// TIA Portal V18 export
FUNCTION "fcFonctionMathLAD" : Void   // FC7, LAD
{ S7_Optimized_Access := 'TRUE' }
// stored: SetENOAutomatically false
   VAR_INPUT
      iInput1 : Bool;
      iInput2 : Bool;
      iInput3 : Bool;
   END_VAR
   VAR_OUTPUT
      oOutput : Bool;
   END_VAR
BEGIN

REGION Network 1
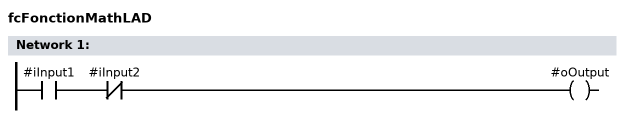
   RUNG wire#powerrail
      Contact( #iInput1 )
      I_Contact( #iInput2 )
      Coil( #oOutput )
   END_RUNG
   // the same network as SCL:
   #oOutput := #iInput1 AND NOT #iInput2;
END_REGION
END_FUNCTION
